// TwinCAT 3 PLC project Tut2_3
// ProgramVersion: 3.1.4023.0
// libraries:
//   Tc2_Standard, * (Beckhoff Automation GmbH)
//   Tc2_System, * (Beckhoff Automation GmbH)
//   Tc3_Module, * (Beckhoff Automation GmbH)
// project tree:
//   / GlobalTextList.TcGTLO, PlcTask.TcTTO, Visualization Manager.TcVMO (not stored)
//   MAIN_POU/ MAIN.TcPOU
//   Virtual controll Box/DUTs/ E_Joy.TcDUT, E_Mode.TcDUT (not stored), E_Status.TcDUT (not stored), ST_BoxParam.TcDUT, ST_VisuParam.TcDUT (not stored)
//   Virtual controll Box/Function_Block/ FB_ModeCBox.TcPOU, FB_ModeSelect.TcPOU, FB_ModeVisu.TcPOU, FB_Status.TcPOU
//   Virtual controll Box/GVLs/ HMI.TcGVL, Input.TcGVL, Output.TcGVL, Parameters.TcGVL
//   Virtual controll Box/Interface/ I_Mode.TcIO (not stored)
//   Virtual controll Box/POUs/ P_VCB.TcPOU
//   VISUs/ VirtualBoxHMI.TcVIS
// real-time tasks:
//   TASK PlcTask: cycle T#10ms, priority 20, ADS port 350
//   TASK PlcTask1: cycle T#10ms, priority 21, ADS port 351

CONFIGURATION Tut2_3
    RESOURCE PLC ON TwinCAT3
        TASK PlcTask(INTERVAL := T#10ms, PRIORITY := 21);
        PROGRAM MAIN WITH PlcTask : MAIN;
    END_RESOURCE
END_CONFIGURATION

// ---- Virtual controll Box/DUTs/E_Joy.TcDUT
{attribute 'qualified_only'}
{attribute 'strict'}
TYPE E_Joy :
(
	Joy_X,
	Joy_Y
);
END_TYPE

// ---- Virtual controll Box/DUTs/ST_BoxParam.TcDUT
TYPE ST_BoxParam :
STRUCT
	bStartPushButton : BOOL;
	bStopPushButton : BOOL;
	bTopSJoy : BOOL;
	fJoy_X : LREAL;
	fJoy_Y : LREAL;
	bManual : BOOL;
	bAuto : BOOL;
END_STRUCT
END_TYPE

// ---- Virtual controll Box/GVLs/HMI.TcGVL
{attribute 'qualified_only'}
VAR_GLOBAL
eStatus : E_Status;
stVisuParam : ST_VisuParam;
eMode : E_Mode;
END_VAR

// ---- Virtual controll Box/GVLs/Input.TcGVL
{attribute 'qualified_only'}
VAR_GLOBAL
	stBoxParam : ST_BoxParam;
	
END_VAR

// ---- Virtual controll Box/GVLs/Output.TcGVL
{attribute 'qualified_only'}
VAR_GLOBAL
	eMode : E_Mode;
END_VAR

// ---- Virtual controll Box/GVLs/Parameters.TcGVL
{attribute 'qualified_only'}
VAR_GLOBAL
	stBoxParam : ST_BoxParam;
END_VAR

// ---- MAIN_POU/MAIN.TcPOU
PROGRAM MAIN
VAR
END_VAR

P_VCB();

END_PROGRAM

// ---- Virtual controll Box/POUs/P_VCB.TcPOU
PROGRAM P_VCB
VAR
	eSwitch : E_Mode;
	fbModeSelect : FB_ModeSelect;
	fbStatus : FB_Status;
END_VAR

fbModeSelect();

fbStatus(
bFault := HMI.stVisuParam.bFault,
bStart:= HMI.stVisuParam.bStart,
bStop := HMI.stVisuParam.bStop,
bRunning := HMI.stVisuParam.bRunning,
eStatus => HMI.eStatus,
bAuto := HMI.stVisuParam.bAuto,
bOn := HMI.stVisuParam.bOn
);

END_PROGRAM

// ---- Virtual controll Box/Function_Block/FB_ModeSelect.TcPOU
FUNCTION_BLOCK FB_ModeSelect
VAR_INPUT
	bControlBox : BOOL;
END_VAR
VAR_OUTPUT
END_VAR
VAR
	fbModeVisu : FB_ModeVisu;
	fbMode : I_Mode := fbModeVisu;
	fbModeCBox: FB_ModeCBox;
END_VAR

IF NOT (bControlBox) THEN
	
fbMode := fbModeVisu;
	IF NOT (HMI.stVisuParam.bOn) THEN
			fbMode.OFF(TRUE);
			fbMode.Auto(FALSE);
			fbMode.Manual(FALSE);
		
	ELSIF (HMI.stVisuParam.bOn) AND NOT (HMI.stVisuParam.bAuto) THEN
			fbMode.OFF(FALSE);
			fbMode.Auto(FALSE);
			fbMode.Manual(TRUE);
		
	ELSIF (HMI.stVisuParam.bOn) AND (HMI.stVisuParam.bAuto) THEN
			fbMode.OFF(FALSE);
			fbMode.Auto(TRUE);
			fbMode.Manual(FALSE);
		
	ELSE
			fbMode.OFF(FALSE);
			fbMode.Auto(FALSE);
			fbMode.Manual(FALSE);
		
	END_IF
	
ELSE
	
	fbMode := fbModeCBox;
	IF NOT (Input.stBoxParam.bAuto) AND NOT(Input.stBoxParam.bManual) THEN
			fbMode.OFF(TRUE);
			fbMode.Auto(FALSE);
			fbMode.Manual(FALSE);
		
	ELSIF NOT (Input.stBoxParam.bAuto) AND Input.stBoxParam.bManual THEN
			fbMode.OFF(FALSE);
			fbMode.Auto(FALSE);
			fbMode.Manual(TRUE);
		
	ELSIF NOT (Input.stBoxParam.bManual) AND Input.stBoxParam.bAuto THEN
			fbMode.OFF(FALSE);
			fbMode.Auto(TRUE);
			fbMode.Manual(FALSE);
		
	ELSE
			fbMode.OFF(FALSE);
			fbMode.Auto(FALSE);
			fbMode.Manual(FALSE);
		
	END_IF
	
END_IF

END_FUNCTION_BLOCK

// ---- Virtual controll Box/Function_Block/FB_ModeVisu.TcPOU
FUNCTION_BLOCK FB_ModeVisu IMPLEMENTS I_Mode
VAR_INPUT
END_VAR
VAR_OUTPUT
END_VAR
VAR
END_VAR

METHOD Auto
VAR_INPUT
	bEnable : BOOL;
END_VAR
IF bEnable THEN 
	HMI.eMode := E_Mode.Auto;
END_IF
END_METHOD

METHOD Manual
VAR_INPUT
	bEnable: BOOL;
END_VAR
IF bEnable THEN 
	HMI.eMode := E_Mode.Manual;
END_IF
END_METHOD

METHOD OFF
VAR_INPUT
	bEnable: BOOL;
END_VAR
IF bEnable THEN 
	HMI.eMode := E_Mode.OFF;
END_IF
END_METHOD

END_FUNCTION_BLOCK

// ---- Virtual controll Box/Function_Block/FB_ModeCBox.TcPOU
FUNCTION_BLOCK FB_ModeCBox IMPLEMENTS I_Mode
VAR_INPUT
END_VAR
VAR_OUTPUT
END_VAR
VAR
END_VAR

METHOD Auto
VAR_INPUT
	bEnable : BOOL;
END_VAR
IF bEnable THEN 
	Output.eMode := E_Mode.Auto;
END_IF
END_METHOD

METHOD Manual
VAR_INPUT
	bEnable : BOOL;
END_VAR
IF bEnable THEN 
	Output.eMode := E_Mode.Manual;
END_IF
END_METHOD

METHOD OFF 
VAR_INPUT
	bEnable : BOOL;
END_VAR
IF bEnable THEN 
	Output.eMode := E_Mode.OFF;
END_IF
END_METHOD

END_FUNCTION_BLOCK

// ---- Virtual controll Box/Function_Block/FB_Status.TcPOU
FUNCTION_BLOCK FB_Status
VAR_INPUT
	bFault : BOOL;
	bStart : BOOL;
	bStop : BOOL;
	bRunning : BOOL;
	bAuto : BOOL;
	bOn : BOOL;
END_VAR
VAR_OUTPUT
	eStatus : E_Status := E_Status.NotReady;
END_VAR
VAR
END_VAR


CASE eStatus OF 

	E_Status.NotReady:
		IF bOn THEN
			eStatus := E_Status.Ready;
		ELSE
			HMI.stVisuParam.bFault := FALSE;
			HMI.stVisuParam.bStop := FALSE;
			eStatus := E_Status.NotReady;
			
			
		END_IF
		
	E_Status.Ready:
		IF bOn THEN
			eStatus := E_Status.Ready;
		ELSE
			eStatus := E_Status.NotReady;
		END_IF
		
		IF bStart THEN
			eStatus := E_Status.Starting;
		END_IF
	
	E_Status.Starting:
			eStatus := E_Status.Running;
		
	E_Status.Running:
		IF bAuto AND bStart AND bOn THEN
			HMI.stVisuParam.bRunning := TRUE;
			eStatus := E_Status.Running;
			
		ELSIF
			bFault THEN
			eStatus := E_Status.Fault;
			
		ELSIF
			 NOT (bAuto) AND bOn THEN
			HMI.stVisuParam.bRunning := TRUE;
			eStatus := E_Status.Running;
				IF bStop THEN
				eStatus := E_Status.Stopping;
				END_IF
		
		
		ELSE
			HMI.stVisuParam.bRunning := FALSE;
			eStatus := E_Status.Ready;
		END_IF
		
		
		
		
	E_Status.Stopping:
		HMI.stVisuParam.bRunning := FALSE;
		bStop := TRUE;
		//Set in a delay to show the stopping longer.
		eStatus := E_Status.NotReady;
	
	E_Status.Fault:
		//Til steget der vi dektekterer fault//eStatus := E_Status.Fault;
		IF bOn THEN	
			HMI.stVisuParam.bStop := TRUE; // LIGHT
			HMI.stVisuParam.bRunning := FALSE;
			eStatus := E_Status.Fault;
		ELSE
			eStatus := E_Status.NotReady;
		END_IF
END_CASE

END_FUNCTION_BLOCK

// ---- GlobalTextList.TcGTLO
TEXTLIST GlobalTextList
  818 = '%0.1f'
  935 = '0.5m'
  892 = '0m'
  175 = 'AUTO'
  667 = 'Auto / Manual'
  104 = 'Boom Angle: %0.1f [deg]'
  58 = 'Current Max Piston Stroke: %0.1f [m] '
  995 = 'Cylinder Position Reference: %f [m]'
  25 = 'Cylinder Velocity Reference: %f [m/s]'
  409 = 'ENABLE'
  527 = 'End Stop Status: %s '
  343 = 'Fault'
  703 = 'Joy_X'
  91 = 'Joy_x'
  757 = 'Joy_Y'
  94 = 'Label'
  660 = 'MANUAL'
  8 = 'Manual Cylinder Position   Reference [m]'
  396 = 'MODE'
  50 = 'Mode: %s'
  76 = 'Mode: %s '
  646 = 'New Max Piston Stroke: %0.1f [m] '
  604 = 'OFF'
  284 = 'ON'
  270 = 'ON / OFF'
  869 = 'PowerON'
  310 = 'RUNNING'
  160 = 'Running'
  695 = 'Set New Value'
  466 = 'Simulation'
  868 = 'START'
  83 = 'Start'
  882 = 'Status : %s'
  173 = 'Status: %s '
  80 = 'Stop'
  880 = 'Stopping / Fault'
  162 = 'Stopping/Fault'
  730 = 'SYSTEM'
  898 = 'SYSTEM STATUS'
  495 = 'Time: %0.1f [s]'
  74 = 'VRBHMI'
  787 = 'WinchOnly'
END_TEXTLIST

// ---- VISUs/VirtualBoxHMI.TcVIS
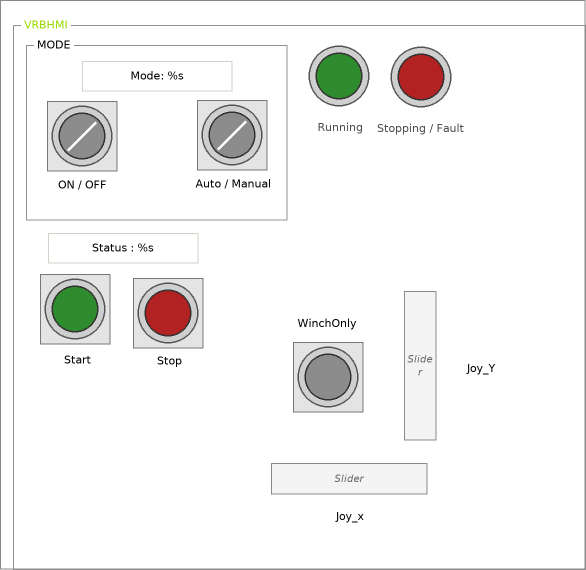
VISUALIZATION VirtualBoxHMI  // 586x570
    GroupBox (13,17 573x553), "VRBHMI"
        PushSwitch (27,257 70x70), variable: HMI.stVisuParam.bStart, behaviour: TAP, style: Switch-PushSwitch-Green
        PushSwitch (120,261 70x70), variable: HMI.stVisuParam.bStop, behaviour: TAP, style: Switch-PushSwitch-Red
        Lamp1 (291,24 70x70), variable: HMI.stVisuParam.bRunning, style: Lamp-Lamp1-Green
        Lamp1 (373,25 70x70), variable: HMI.stVisuParam.bStop, style: Lamp-Lamp1-Red
        Slider (5682,5127 161x29), scale 0..100
        Slider (5815,4955 30x143), scale 0..100
        Label (5690,5182 150x30), "Joy_X"
        Label (5852,4969 65x118), "Joy_Y"
        Label (360,97 95x29), "Stopping / Fault"
        Label (105,330 103x28), "Stop"
        Label (19,328 91x30), "Start"
        GroupBox (13,20 261x183), "MODE"
            Label (11,133 91x30), "ON / OFF"
            RotarySwitch (171,63 70x70), variable: HMI.stVisuParam.bAuto, behaviour: TOGGLE, style: Switch-RotarySwitch-Gray
            Label (162,132 91x30), "Auto / Manual"
            Textfield (56,24 150x30), "Mode: %s", text variable: HMI.eMode
            RotarySwitch (21,64 70x70), variable: HMI.stVisuParam.bOn, behaviour: TOGGLE, style: Switch-RotarySwitch-Gray
        Textfield (35,216 150x30), "Status : %s", text variable: HMI.eStatus
        Label (193,329 103x28)
        Label (280,96 95x29), "Running"
        Slider (258,446 156x31), variable: HMI.stVisuParam.fJoy_X, scale -1..1
        Slider (391,274 32x149), variable: HMI.stVisuParam.fJoy_Y, scale -1..1
        Label (298,484 78x31), "Joy_x"
        Label (433,338 70x27), "Joy_Y"
        PushSwitch (280,325 70x70), variable: HMI.stVisuParam.bTopSwitchJoy, behaviour: TOGGLE, style: Switch-PushSwitch-Gray
        Label (279,293 70x27), "WinchOnly"
END_VISUALIZATION
